(* IEC 61131-3 sources: b-rformacion/controladorTemperaturas, 2 files *)

(* ---- Main.st ---- *)
//Autor : Erik Churo
//Descripcion : programa que realiza el control de temperatura
//este control es vital, ejecutar cada 10ms
PROGRAM _INIT

END_PROGRAM

PROGRAM _CYCLIC
	//control de temperatura
	IF ai_temperatura_real <= ai_temperatura_minima THEN //temperatura igual o inferior a la temperatura minima
		ao_alarma := 'Tş BAJA'; //mensaje de error, temperatura no suficiente
	ELSIF ai_temperatura_real >= ai_temperatura_maxima THEN //temperatura igual o superior a la temperatura maxima
		ao_alarma := 'Tş ALTA';//mensaje de error, temperatura excesiva
	ELSE ////temperatura correcta
		ao_alarma := 'Tş OK'; //mensaje de acierto
	END_IF
END_PROGRAM

(* ---- Variables.var ---- *)
VAR
	ai_temperatura_minima : {REDUND_UNREPLICABLE} REAL := 50.0; (*Temperatura minima*)
	ai_temperatura_maxima : {REDUND_UNREPLICABLE} REAL := 150.0; (*Temperatura maxima*)
	ao_alarma : STRING[7]; (*Feedback*)
END_VAR
